// Mitsubishi GX Works2 project: 짝수,홀수   PLC: Q02/Q02H

PROGRAM MAIN
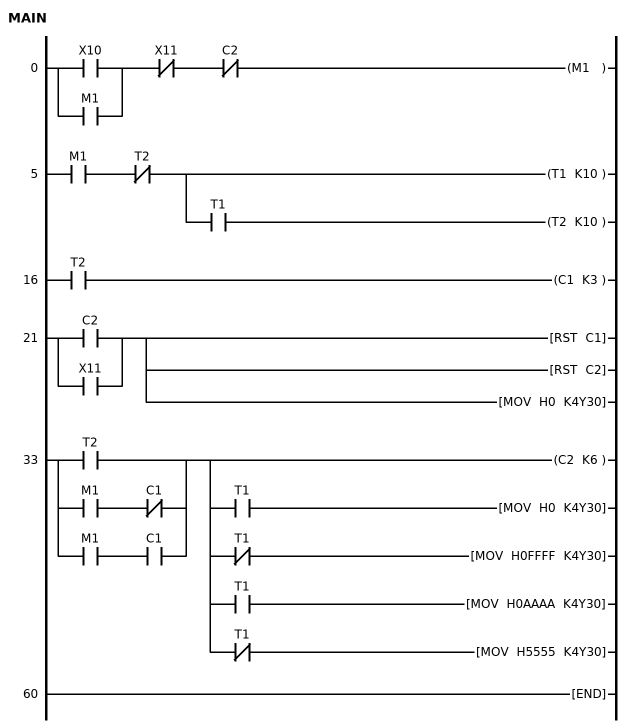
0     LD      X10
      OR      M1
      ANI     X11
      ANI     C2
      OUT     M1
5     LD      M1
      ANI     T2
      OUT     T1 K10
      AND     T1
      OUT     T2 K10
16    LD      T2
      OUT     C1 K3
21    LD      C2
      OR      X11
      RST     C1
      RST     C2
      MOV     H0 K4Y30
33    LD      T2
      LD      M1
      ANI     C1
      ORB
      LD      M1
      AND     C1
      ORB
      OUT     C2 K6
      MPS
      AND     T1
      MOV     H0 K4Y30
      MRD
      ANI     T1
      MOV     H0FFFF K4Y30
      MRD
      AND     T1
      MOV     H0AAAA K4Y30
      MPP
      ANI     T1
      MOV     H5555 K4Y30
60    END
END_PROGRAM
